// TIA Portal project "MTU_Bauteilträger(BTTR)_V16" (V16)

(* hardware
DEVICE "ET 200SP station_1"  ET 200SP-Station
   slot 0: "Rack_0"  Rack  6ES5 710-8MAx1
   slot 1: "-33K1"  CPU 1512SP F-1 PN  6ES7 512-1SK01-0AB0  V2.8
      slot 32768: "PROFINET interface_1"  X1
   slot 2: "-33K2"  DI 16x24VDC ST  6ES7 131-6BH01-0BA0  V0.0
      slot 1: "-33K2"  DI 16x24VDC ST
   slot 3: "-33K3"  DI 16x24VDC ST  6ES7 131-6BH01-0BA0  V0.0
      slot 1: "-33K3"  DI 16x24VDC ST
   slot 4: "-33K5"  DQ 4x24VDC/2A ST  6ES7 132-6BD20-0BA0  V1.1
      slot 1: "-33K5"  DQ 4x24VDC/2A ST
   slot 5: "-33K6"  DQ 4x24VDC/2A ST  6ES7 132-6BD20-0BA0  V1.1
      slot 1: "-33K6"  DQ 4x24VDC/2A ST
   slot 6: "Server module_1"  Server module  6ES7 193-6PA00-0AA0  V1.1
      slot 1: "Server module_1"  Server module
   slot 127: "BA 2xRJ45"  BA 2xRJ45  6ES7 193-6AR00-0AA0  V0.0
      slot 32769: "Port_1"  6ES7 193-6AR00-0AA0
      slot 32770: "Port_2"  6ES7 193-6AR00-0AA0
DEVICE "-55K1"  PnPn.Device
   slot 0: "Rack"  Rail  1.0
   slot 0: "pn-pn-coupler.X1"  PN/PN Coupler  6ES7 158-3AD10-0XA0  V4.2
   slot 1: "pn-pn-coupler"  PN/PN Coupler  6ES7 158-3AD10-0XA0  V4.2
   slot 127: "BA 2xRJ45"  BA 2xRJ45  6ES7 193-6AR00-0AA0  V0.0
      slot 1: "Port_1"  X1 P1 R  6ES7 193-6AR00-0AA0  V0.0
      slot 2: "Port_2"  X1 P2 R  6ES7 193-6AR00-0AA0  V0.0
   slot 127: "BA 2xRJ45"  BA 2xRJ45  6ES7 193-6AR00-0AA0  V0.0
      slot 1: "Port_1"  X2 P1 R  6ES7 193-6AR00-0AA0  V0.0
      slot 2: "Port_2"  X2 P2 R  6ES7 193-6AR00-0AA0  V0.0
*)

// ===== PLC "-33K1"  CPU 1512SP F-1 PN =====

VAR_GLOBAL   // PLC tag table "Default tag table"
   "System_Byte" AT %MB1 : Byte;
   "FirstScan" AT %M1.0 : Bool;
   "DiagStatusUpdate" AT %M1.1 : Bool;
   "AlwaysTRUE" AT %M1.2 : Bool;
   "AlwaysFALSE" AT %M1.3 : Bool;
   "System_Byte(1)" AT %MB1 : Byte;
   "Clock_Byte" AT %MB0 : Byte;
   "Clock_10Hz" AT %M0.0 : Bool;
   "Clock_5Hz" AT %M0.1 : Bool;
   "Clock_2.5Hz" AT %M0.2 : Bool;
   "Clock_2Hz" AT %M0.3 : Bool;
   "Clock_1.25Hz" AT %M0.4 : Bool;
   "Clock_1Hz" AT %M0.5 : Bool;
   "Clock_0.625Hz" AT %M0.6 : Bool;
   "Clock_0.5Hz" AT %M0.7 : Bool;
END_VAR

VAR_GLOBAL   // PLC tag table "Ausgänge"
   "O_BTTR1_UnlockComp" AT %Q1610.0 : Bool;   // Bauteilträger 1 Bauteil entriegeln (1=entriegeln)
   "O_BTTR2_UnlockComp" AT %Q1610.1 : Bool;   // Bauteilträger 2 Bauteil entriegeln (1=entriegeln)
   "O_BTTR3_UnlockComp" AT %Q1610.2 : Bool;   // Bauteilträger 3 Bauteil entriegeln (1=entriegeln)
   "O_BTTR4_UnlockComp" AT %Q1610.3 : Bool;   // Bauteilträger 4 Bauteil entriegeln (1=entriegeln)
   "O_BTTR5_UnlockComp" AT %Q1611.0 : Bool;   // Bauteilträger 5 Bauteil entriegeln (1=entriegeln)
   "O_BTTR6_UnlockComp" AT %Q1611.1 : Bool;   // Bauteilträger 6 Bauteil entriegeln (1=entriegeln)
   "A1611.2" AT %Q1611.2 : Bool;   // Reserve
   "A1611.3" AT %Q1611.3 : Bool;   // Reserve
END_VAR

VAR_GLOBAL   // PLC tag table "Eingänge"
   "I_BTTR1_CompMon" AT %I1610.0 : Bool;   // Bauteilträger 1 INS Bauteilüberwachung (0=Platz leer/1=Platz belegt)
   "I_BTTR1_CompLock_SW1" AT %I1610.1 : Bool;   // Bauteilträger 1 RM Bauteilverriegelung Schalter 1
   "I_BTTR1_CompLock_SW2" AT %I1610.2 : Bool;   // Bauteilträger 1 RM Bauteilverriegelung Schalter 2
   "E1610.3" AT %I1610.3 : Bool;   // Bauteilträger 1 Reserve
   "I_BTTR2_CompMon" AT %I1610.4 : Bool;   // Bauteilträger 2 INS Bauteilüberwachung (0=Platz leer/1=Platz belegt)
   "I_BTTR2_CompLock_SW1" AT %I1610.5 : Bool;   // Bauteilträger 2 RM Bauteilverriegelung Schalter 1
   "I_BTTR2_CompLock_SW2" AT %I1610.6 : Bool;   // Bauteilträger 2 RM Bauteilverriegelung Schalter 2
   "E1610.7" AT %I1610.7 : Bool;   // Bauteilträger 2 Reserve
   "I_BTTR3_CompMon" AT %I1611.0 : Bool;   // Bauteilträger 3 INS Bauteilüberwachung (0=Platz leer/1=Platz belegt)
   "I_BTTR3_CompLock_SW1" AT %I1611.1 : Bool;   // Bauteilträger 3 RM Bauteilverriegelung Schalter 1
   "I_BTTR3_CompLock_SW2" AT %I1611.2 : Bool;   // Bauteilträger 3 RM Bauteilverriegelung Schalter 2
   "E1611.3" AT %I1611.3 : Bool;   // Bauteilträger 3 Reserve
   "I_BTTR4_CompMon" AT %I1611.4 : Bool;   // Bauteilträger 4 INS Bauteilüberwachung (0=Platz leer/1=Platz belegt)
   "I_BTTR4_CompLock_SW1" AT %I1611.5 : Bool;   // Bauteilträger 4 RM Bauteilverriegelung Schalter 1
   "I_BTTR4_CompLock_SW2" AT %I1611.6 : Bool;   // Bauteilträger 4 RM Bauteilverriegelung Schalter 2
   "E1611.7" AT %I1611.7 : Bool;   // Bauteilträger 4 Reserve
   "I_BTTR5_CompMon" AT %I1612.0 : Bool;   // Bauteilträger 5 INS Bauteilüberwachung (0=Platz leer/1=Platz belegt)
   "I_BTTR5_CompLock_SW1" AT %I1612.1 : Bool;   // Bauteilträger 5 RM Bauteilverriegelung Schalter 1
   "I_BTTR5_CompLock_SW2" AT %I1612.2 : Bool;   // Bauteilträger 5 RM Bauteilverriegelung Schalter 2
   "E1612.3" AT %I1612.3 : Bool;   // Bauteilträger 5 Reserve
   "I_BTTR6_CompMon" AT %I1612.4 : Bool;   // Bauteilträger 6 INS Bauteilüberwachung (0=Platz leer/1=Platz belegt)
   "I_BTTR6_CompLock_SW1" AT %I1612.5 : Bool;   // Bauteilträger 6 RM Bauteilverriegelung Schalter 1
   "I_BTTR6_CompLock_SW2" AT %I1612.6 : Bool;   // Bauteilträger 6 RM Bauteilverriegelung Schalter 2
   "E1612.7" AT %I1612.7 : Bool;   // Bauteilträger 6 Reserve
   "I_TankLevel_75" AT %I1613.0 : Bool;   // Tanküberwachung Füllstand >=75% (0=>=75%/1=<=75%)
   "E1613.1" AT %I1613.1 : Bool;   // Tanküberwachung Füllstand >=75% Reserve
   "I_TankLevel_100" AT %I1613.2 : Bool;   // Tanküberwachung Füllstand >=100% (0=>=100%/1=<=100%)
   "E1613.3" AT %I1613.3 : Bool;   // Tanküberwachung Füllstand >=100% Reserve
   "E1613.4" AT %I1613.4 : Bool;   // Reserve
   "E1613.5" AT %I1613.5 : Bool;   // Reserve
   "E1613.6" AT %I1613.6 : Bool;   // Reserve
   "E1613.7" AT %I1613.7 : Bool;   // Reserve
END_VAR

TYPE "UDT_BTTR"
   STRUCT
      ID : DInt;   // Aktuelle Nummer vom Bild
      ESF_ID : DInt;   // Nummer für die Textliste für Zylindernamen
      ESF_Nr : DInt;   // angewählte ESF in der HMI
      Ctrl : Struct
         Unlock : Bool;   // Command to unlock
         Reset_error : Bool;   // Command to reset error
      END_STRUCT;
      Status : Struct
         UnLocked : Bool;   // State (1- unlocked, 0 - locked)
         ErrorBit : Bool;   // Error flag
         ErrorByte : Byte;   // Error type
      END_STRUCT;
   END_STRUCT;
END_TYPE

TYPE "UDT_FM_Bits"
VERSION : 0.1
   STRUCT
      SM : Array[1..2048] of Bool;
   END_STRUCT;
END_TYPE

// folder: Sensor

TYPE "UDT_T_Sensor"
   STRUCT
      Rohsignal : Bool;   // Direkt vom Eingangsignal
      Frei : Bool;   // Sensor frei
      Belegt : Bool;   // Sensor belegt
      T_Frei : Bool;   // Sensor mit T-Zeit frei
      T_Belegt : Bool;   // Senssor mit T-zeit belegt
      T_Dauer_Belegt : Bool;
      Fehler : Bool;   // Fehler aktiv
      Status : Byte;   // 0 = OK 1 = nicht frei 2=nicht belegt
      Temp_Fehler : Struct   // Fehler generieren und wird automatisch im Sensorbaustein zurückgesetzt
         Nicht_frei : Bool;   // Fehler Sensor nicht frei
         Nicht_belegt : Bool;   // Fehler Sensor nicht belegt
      END_STRUCT;
      Setup : Struct
         T_Frei : Time := T#100MS;
         T_Belegt : Time := T#100MS;
         T_Dauer : Time := T#10S;
         Typ : Bool;   // 0 = S 1 = Ö
         Mode : Byte;
      END_STRUCT;
   END_STRUCT;
END_TYPE

TYPE "UDTFltFbStructSeqSK"
   STRUCT
      Aktiv : Byte;   // 1=Aktiv
      Msg : Byte;   // 1=FLT 2=Warn 10=Clear
      StepNo : Int;
      FltID : DInt;
      DeviceID : DInt;
      Station : DInt;
      DeviceText : String[20];
   END_STRUCT;
END_TYPE

// folder: DBs

DATA_BLOCK "DB_Sensors"   // DB1
{ S7_Optimized_Access := 'TRUE' }
VERSION : 0.1
   VAR
      "Sens_BTTR1-11BG1" : "UDT_T_Sensor";   // Bauteilträger 1 INS Bauteilüberwachung (0=Platz leer/1=Platz belegt)
      "Sens_BTTR2-13BG1" : "UDT_T_Sensor";   // Bauteilträger 2 INS Bauteilüberwachung (0=Platz leer/1=Platz belegt)
      "Sens_BTTR3-15BG1" : "UDT_T_Sensor";   // Bauteilträger 3 INS Bauteilüberwachung (0=Platz leer/1=Platz belegt)
      "Sens_BTTR4-17BG1" : "UDT_T_Sensor";   // Bauteilträger 4 INS Bauteilüberwachung (0=Platz leer/1=Platz belegt)
      "Sens_BTTR5-19BG1" : "UDT_T_Sensor";   // Bauteilträger 5 INS Bauteilüberwachung (0=Platz leer/1=Platz belegt)
      "Sens_BTTR6-21BG1" : "UDT_T_Sensor";   // Bauteilträger 6 INS Bauteilüberwachung (0=Platz leer/1=Platz belegt)
      "Sens_UGBTTR-23A1" : "UDT_T_Sensor";   // Tank Untergestell Füllstand >=75%
      "Sens_UGBTTR-23A2" : "UDT_T_Sensor";   // Tank Untergestell Füllstand >=100%
   END_VAR
BEGIN
END_DATA_BLOCK

DATA_BLOCK "DB_M1_SM"   // DB2
{ S7_Optimized_Access := 'TRUE' }
VERSION : 0.1
   VAR
      SM : "UDT_FM_Bits";
      SM_Byte : Array[1..2048] of Byte;
      SM_DInt : Array[1..2048] of DInt;
      SM_Word_Komm : Array[1..100] of Word;
   END_VAR
BEGIN
END_DATA_BLOCK

DATA_BLOCK "DB_BTTR"   // DB4
{ S7_Optimized_Access := 'TRUE' }
VERSION : 0.1
   VAR
      "BTTR1-11K1" : "UDT_BTTR";   // elektr. mag. Verriegelungseinheit Bauteilträger1
      "BTTR2-13K1" : "UDT_BTTR";   // elektr. mag. Verriegelungseinheit Bauteilträger2
      "BTTR3-15K1" : "UDT_BTTR";   // elektr. mag. Verriegelungseinheit Bauteilträger3
      "BTTR4-17K1" : "UDT_BTTR";   // elektr. mag. Verriegelungseinheit Bauteilträger4
      "BTTR5-19K1" : "UDT_BTTR";   // elektr. mag. Verriegelungseinheit Bauteilträger5
      "BTTR6-21K1" : "UDT_BTTR";   // elektr. mag. Verriegelungseinheit Bauteilträger6
   END_VAR
BEGIN
END_DATA_BLOCK

DATA_BLOCK "DB_SPS-BTTR_ProfinetComm"   // DB6
{ S7_Optimized_Access := 'TRUE' }
VERSION : 0.1
   VAR
      DataIn : Struct   // XXX_to_SPS(BTTR/MAG)
         robotSafeArea : Bool;   // Robot out of magazin-area
         enableMagazinMotion : Bool;   // Magazin allowed to turn
         requestIdentification : Bool;   // Identification of loaded parts requested
         robotDoor1Open : Bool;   // Command to open robot-door amr
         robotDoor1Close : Bool;   // Command to close robot-door amr
         robotDoor2Open : Bool;   // Command to open robot-door fix
         robotDoor2Close : Bool;   // Command to close robot-door fix
         "Bit0.7" : Bool;
         requestUndock : Bool;   // Request from AMR to undock
         requestCommunication : Bool;   // Request from PN-Station to take masterpart on communication
         "Bit1.2" : Bool;
         "Bit1.3" : Bool;
         "Bit1.4" : Bool;
         "Bit1.5" : Bool;
         unlockBTTRRequest : Bool;   // Request from Robot to unlock BTTR
         resetBTTRerror : Bool;   // To reset BTTR errors
         requestPlace : UInt;   // Byte2 - Requested place to move
         requestLevel : UInt;   // Byte4 - Requested level for postion to move
         requestPosition : UInt;   // Byte6 - Requested positin to move
         requestSide : UInt;   // Byte8 - Requested place to move on requested side
         Byte10 : Byte;   // Byte10
         Byte11_1 : Byte;   // Byte11
         Byte12_1 : Byte;   // Byte12
         Byte13_1 : Byte;   // Byte13
         Byte14_1 : Byte;   // Byte14
         Byte15_1 : Byte;   // Byte15
         Byte16_1 : Byte;   // Byte16
         Byte17_1 : Byte;   // Byte17
         Byte18_1 : Byte;   // Byte18
         Byte19_1 : Byte;   // Byte19
         Byte20_1 : Byte;   // Byte20
         Byte21_1 : Byte;   // Byte21
         Byte22_1 : Byte;   // Byte22
         Byte23_1 : Byte;   // Byte23
         Byte24_1 : Byte;   // Byte24
         Byte25_1 : Byte;   // Byte25
         Byte26_1 : Byte;   // Byte26
         Byte27_1 : Byte;   // Byte27
         Byte28_1 : Byte;   // Byte28
         Byte29_1 : Byte;   // Byte29
         Byte30_1 : Byte;   // Byte30
         Byte31_1 : Byte;   // Byte10
         Byte32_1 : Byte;   // Byte10
         Byte33_1 : Byte;   // Byte10
         Byte34_1 : Byte;   // Byte10
         Byte35_1 : Byte;   // Byte10
         Byte36_1 : Byte;   // Byte10
         Byte37_1 : Byte;   // Byte10
         Byte38_1 : Byte;   // Byte10
         Byte39_1 : Byte;   // Byte10
         Byte40_1 : Byte;   // Byte10
         Byte41_1 : Byte;   // Byte10
         Byte42_1 : Byte;   // Byte10
         Byte43_1 : Byte;   // Byte10
         Byte44_1 : Byte;   // Byte10
         Byte45_1 : Byte;   // Byte10
         Byte46_1 : Byte;   // Byte10
         Byte47_1 : Byte;   // Byte10
         Byte48_1 : Byte;   // Byte10
         Byte49_1 : Byte;   // Byte10
         Byte50_1 : Byte;   // Byte10
         Byte51_1 : Byte;   // Byte10
         Byte52_1 : Byte;   // Byte10
         Byte53_1 : Byte;   // Byte10
         Byte54_1 : Byte;   // Byte10
         Byte55_1 : Byte;   // Byte10
         Byte56_1 : Byte;   // Byte10
         Byte57_1 : Byte;   // Byte10
         Byte58_1 : Byte;   // Byte10
         Byte59_1 : Byte;   // Byte10
         Byte60_1 : Byte;   // Byte10
         Byte61_1 : Byte;   // Byte10
         Byte62_1 : Byte;   // Byte10
         Byte63_1 : Byte;   // Byte10
      END_STRUCT;
      DataOut : Struct   // SPS(BTTR/MAG)_to_XXX
         placeDone : Bool;   // Signal indicating moving on requested place done
         enableRobotAccess1 : Bool;   // Signal indicating access for robot amr enabled
         enableRobotAccess2 : Bool;   // Signal indicating access for robot fix enabled
         "Bit0.3" : Bool;
         "Bit0.4" : Bool;
         "Bit0.5" : Bool;
         "Bit0.6" : Bool;
         "Bit0.7" : Bool;
         readyForUndock : Bool;   // Signal indicating magazin is ready to undock
         "Bit1.1" : Bool;
         "Bit1.2" : Bool;
         "Bit1.3" : Bool;
         "Bit1.4" : Bool;
         "Bit1.5" : Bool;
         "Bit1.6" : Bool;
         "Bit1.7" : Bool;
         state : Word;   // Byte2-3
         errorIndication : Word;   // Byte4-5
         placeNbrAct : UInt;   // Byte6-7
         zlr : String[16];   // Byte8-25 - serial number of PLC
         sanr : String[16] := 'BTTR';   // Byte26-43
         InductiveBTTRsensor : Word;   // Byte44-45 (six first bits for six sensors)
         BTTRerror : Word;   // Byte46-47 (six first bits for six BTTR)
         BTTRunlocked : Bool;   // Bit48.0 (BTTR1…6 are unlocked )
         level_75 : Bool;   // Bit48.1 (Tank monitoring level> = 75%)
         level_100 : Bool;   // Bit48.2 (Tank monitoring level> = 100%)
         "Bit48.3" : Bool;
         "Bit48.4" : Bool;
         "Bit48.5" : Bool;
         "Bit48.6" : Bool;
         "Bit48.7" : Bool;
         Byte49 : Byte;
         Byte50 : Byte;
         Byte51 : Byte;
         Byte52 : Byte;
         Byte53 : Byte;
         Byte54 : Byte;
         Byte55 : Byte;
         Byte56 : Byte;
         Byte57 : Byte;
         Byte58 : Byte;
         Byte59 : Byte;
         Byte60 : Byte;
         Byte61 : Byte;
         Byte62 : Byte;
         Byte63 : Byte;
      END_STRUCT;
      StatusRead : DWord;
      StatusWrite : DWord;
      LengthRead : Int;
   END_VAR
BEGIN
END_DATA_BLOCK

// folder: Instances

DATA_BLOCK "Sensors_DB"   // DB3
{ S7_Optimized_Access := 'TRUE' }
VERSION : 0.1
// stored: InstanceOfName ESF_Sensors
"ESF_Sensors"
BEGIN
END_DATA_BLOCK

DATA_BLOCK "ESF_BTTR_DB"   // DB5
{ S7_Optimized_Access := 'TRUE' }
VERSION : 0.1
// stored: InstanceOfName ESF_BTTR
"ESF_BTTR"
BEGIN
END_DATA_BLOCK

DATA_BLOCK "BTTR_Control_DB"   // DB7
{ S7_Optimized_Access := 'TRUE' }
VERSION : 0.1
// stored: InstanceOfName BTTR_Control
"BTTR_Control"
BEGIN
END_DATA_BLOCK

// folder: (top level)

FUNCTION_BLOCK "ESF_Sensors"   // FB1, SCL
{ S7_Optimized_Access := 'TRUE' }
VERSION : 0.1
   VAR
      "Sens_BTTR1-11BG1" : "FB_T_Sensor";
      "Sens_BTTR2-13BG1" : "FB_T_Sensor";
      "Sens_BTTR3-15BG1" : "FB_T_Sensor";
      "Sens_BTTR4-17BG1" : "FB_T_Sensor";
      "Sens_BTTR5-19BG1" : "FB_T_Sensor";
      "Sens_BTTR6-21BG1" : "FB_T_Sensor";
      "Sens_UGBTTR-23A1" : "FB_T_Sensor";
      "Sens_UGBTTR-23A2" : "FB_T_Sensor";
   END_VAR
BEGIN
   (*##############################################################################################################################*)
   (*                                                 FunctionBlock Description                                                    *)
   (*##############################################################################################################################*)
   (*################################################################################################################################
   Created by: preccon Robotics
   Department: 
   Creator: d.shulgin
   Creation Date: 2021-09-24
   Version: V1.0.0.0
   Function Description:
       Inputs:
           --NONE--
           Description in IO table
       Outputs:
           --NONE--
           Description in IO table
       Function:
           Creating sensors instances  

   Last Changed:
       2021-09-24 d.shulgin: V1.0.0.0 Created FunctionBlock

   ################################################################################################################################*)



   REGION Bauteilträger 1 INS Bauteilüberwachung
      #"Sens_BTTR1-11BG1"(E_Sensor:="I_BTTR1_CompMon",
                          SensorMode:=0,
                          Error => "DB_M1_SM".SM.SM[501],//flag of error [size - bool]
                          "ErrorState" => "DB_M1_SM".SM_Byte[501],//type of error [size - byte]
                          Sensor:="DB_Sensors"."Sens_BTTR1-11BG1");
   END_REGION

   REGION Bauteilträger 2 INS Bauteilüberwachung
       #"Sens_BTTR2-13BG1"(E_Sensor:="I_BTTR2_CompMon",
                           SensorMode:=0,
                           Error => "DB_M1_SM".SM.SM[502],
                           "ErrorState" => "DB_M1_SM".SM_Byte[502],
                           Sensor:="DB_Sensors"."Sens_BTTR2-13BG1");
   END_REGION

   REGION Bauteilträger 3 INS Bauteilüberwachung
       #"Sens_BTTR3-15BG1"(E_Sensor:="I_BTTR3_CompMon",
                           SensorMode:=0,
                           Error => "DB_M1_SM".SM.SM[503],
                           "ErrorState" => "DB_M1_SM".SM_Byte[503],
                           Sensor:="DB_Sensors"."Sens_BTTR3-15BG1");
   END_REGION

   REGION Bauteilträger 4 INS Bauteilüberwachung
       #"Sens_BTTR4-17BG1"(E_Sensor:="I_BTTR4_CompMon",
                           SensorMode:=0,
                           Error => "DB_M1_SM".SM.SM[504],
                           "ErrorState" => "DB_M1_SM".SM_Byte[504],
                           Sensor:="DB_Sensors"."Sens_BTTR4-17BG1");
   END_REGION

   REGION Bauteilträger 5 INS Bauteilüberwachung
       #"Sens_BTTR5-19BG1"(E_Sensor:="I_BTTR5_CompMon",
                           SensorMode:=0,
                           Error => "DB_M1_SM".SM.SM[505],
                           "ErrorState" => "DB_M1_SM".SM_Byte[505],
                           Sensor:="DB_Sensors"."Sens_BTTR5-19BG1");
   END_REGION

   REGION Bauteilträger 6 INS Bauteilüberwachung
       #"Sens_BTTR6-21BG1"(E_Sensor:="I_BTTR6_CompMon",
                           SensorMode:=0,
                           Error => "DB_M1_SM".SM.SM[506],
                           "ErrorState" => "DB_M1_SM".SM_Byte[506],
                           Sensor:="DB_Sensors"."Sens_BTTR6-21BG1");
   END_REGION


   REGION Tanküberwachung Füllstand >=75% (0=>=75%/1=<=75%)
       #"Sens_UGBTTR-23A1"(E_Sensor := "I_TankLevel_75",
                           SensorMode := 0,
                           Error => "DB_M1_SM".SM.SM[507],
                           "ErrorState" => "DB_M1_SM".SM_Byte[507],
                           Sensor := "DB_Sensors"."Sens_UGBTTR-23A1");
   END_REGION

   REGION Tanküberwachung Füllstand >=100% (0=>=100%/1=<=100%)
       #"Sens_UGBTTR-23A2"(E_Sensor:="I_TankLevel_100",
                           SensorMode:=0,
                           Error => "DB_M1_SM".SM.SM[508],
                           "ErrorState" => "DB_M1_SM".SM_Byte[508],
                           Sensor:="DB_Sensors"."Sens_UGBTTR-23A2");
   END_REGION
END_FUNCTION_BLOCK

FUNCTION_BLOCK "ESF_BTTR"   // FB3, SCL
{ S7_Optimized_Access := 'TRUE' }
VERSION : 0.1
   VAR
      BTTR1 : "FB_BTTR_Ctrl";
      BTTR2 : "FB_BTTR_Ctrl";
      BTTR3 : "FB_BTTR_Ctrl";
      BTTR4 : "FB_BTTR_Ctrl";
      BTTR5 : "FB_BTTR_Ctrl";
      BTTR6 : "FB_BTTR_Ctrl";
   END_VAR
BEGIN
   (*##############################################################################################################################*)
   (*                                                 FunctionBlock Description                                                    *)
   (*##############################################################################################################################*)
   (*################################################################################################################################
   Created by: preccon Robotics
   Department: 
   Creator: d.shulgin
   Creation Date: 2021-09-24
   Version: V1.0.0.0
   Function Description:
       Inputs:
           --NONE--
           Description in IO table
       Outputs:
           --NONE--
           Description in IO table
       Function:
           Creating 6 instances for 6 BTTR units 

   Last Changed:
       2021-09-24 d.shulgin: V1.0.0.0 Created FunctionBlock

   ################################################################################################################################*)


   REGION BTTR1-11K1
   #BTTR1(Verr_Unlock:=FALSE,
          Freigabe:=TRUE,
          E_Schalter1:="I_BTTR1_CompLock_SW1",
          E_Schalter2:="I_BTTR1_CompLock_SW2",
          A_BTTR_Unlock=>"O_BTTR1_UnlockComp",
          BTTR:="DB_BTTR"."BTTR1-11K1");

   END_REGION

   REGION BTTR2-13K1
       #BTTR2(Verr_Unlock:=FALSE,
              Freigabe:=TRUE,
              E_Schalter1:="I_BTTR2_CompLock_SW1",
              E_Schalter2:="I_BTTR2_CompLock_SW2",
              A_BTTR_Unlock=>"O_BTTR2_UnlockComp",
              BTTR:="DB_BTTR"."BTTR2-13K1");

   END_REGION

   REGION BTTR3-15K1
       #BTTR3(Verr_Unlock:=FALSE,
              Freigabe:=TRUE,
              E_Schalter1:="I_BTTR3_CompLock_SW1",
              E_Schalter2:="I_BTTR3_CompLock_SW2",
              A_BTTR_Unlock=>"O_BTTR3_UnlockComp",
              BTTR:="DB_BTTR"."BTTR3-15K1");

   END_REGION

   REGION BTTR4-17K1
       #BTTR4(Verr_Unlock:=FALSE,
              Freigabe:=TRUE,
              E_Schalter1:="I_BTTR4_CompLock_SW1",
              E_Schalter2:="I_BTTR4_CompLock_SW2",
              A_BTTR_Unlock=>"O_BTTR4_UnlockComp",
              BTTR:="DB_BTTR"."BTTR4-17K1");

   END_REGION

   REGION BTTR5-19K1
       #BTTR5(Verr_Unlock:=FALSE,
              Freigabe:=TRUE,
              E_Schalter1:="I_BTTR5_CompLock_SW1",
              E_Schalter2:="I_BTTR5_CompLock_SW2",
              A_BTTR_Unlock=>"O_BTTR5_UnlockComp",
              BTTR:="DB_BTTR"."BTTR5-19K1");

   END_REGION

   REGION BTTR6-21K1
       #BTTR6(Verr_Unlock:=FALSE,
              Freigabe:=TRUE,
              E_Schalter1:="I_BTTR6_CompLock_SW1",
              E_Schalter2:="I_BTTR6_CompLock_SW2",
              A_BTTR_Unlock=>"O_BTTR6_UnlockComp",
              BTTR:="DB_BTTR"."BTTR6-21K1");

   END_REGION
END_FUNCTION_BLOCK

FUNCTION_BLOCK "BTTR_Control"   // FB4, SCL
{ S7_Optimized_Access := 'TRUE' }
VERSION : 0.1
   VAR
      GETIO_Instance : GETIO;   // Profinet IO interface READ
      SETIO_Instance : SETIO;   // Profinet IO interface WRITE
      GET_IM_DATA_Instance : Get_IM_Data;
      bGetImDataDONE : Bool;
      imData : IM0_Data;
   END_VAR
BEGIN
   (*##############################################################################################################################*)
   (*                                                 FunctionBlock Description                                                    *)
   (*##############################################################################################################################*)
   (*################################################################################################################################
   Created by: preccon Robotics
   Department: 
   Creator: d.shulgin
   Creation Date: 2021-09-24
   Version: V1.0.0.0
   Function Description:
       Inputs:
           --NONE--
           Description in IO table
       Outputs:
           --NONE--
           Description in IO table
       Function:
           Read/Write profinet IO-signals beatween BTTR and AMR CS9 

   Last Changed:
       2021-09-24 d.shulgin: V1.0.0.0 Created FunctionBlock
       2021-10-04 d.shulgin: inverse signals from sensors "Bauteilträger Bauteilüberwachung"
       2021-10-06 d.shulgin: Updating signals in "DB_SPS-BTTR_ProfinetComm[DB6]"
       2021-10-08 d.shulgin: Adding reading serial number function
       2021-10-12 d.shulgin: Adding pn-pn Coupler
       2021-10-12 d.shulgin: Updating signals in "DB_SPS-BTTR_ProfinetComm[DB6]"

   ################################################################################################################################*)



   REGION Init
       //Read PLC serial number
       #GET_IM_DATA_Instance(LADDR:="Local",
                             IM_TYPE:=0,
                             DONE=>#bGetImDataDONE,
                             DATA:=#imData);

       IF #bGetImDataDONE THEN
           "DB_SPS-BTTR_ProfinetComm".DataOut.zlr:=#imData.Serial_Number;
       END_IF;
   END_REGION


   REGION READ Profinet IO signals
       #GETIO_Instance(ID:="pn-pn-coupler_X1~PROFINET_interface_X1~Rob_toPLC",
                       STATUS=>"DB_SPS-BTTR_ProfinetComm".StatusRead,
                       LEN=>"DB_SPS-BTTR_ProfinetComm".LengthRead,
                       INPUTS:="DB_SPS-BTTR_ProfinetComm".DataIn);

   END_REGION


   REGION Control BTTR
       "DB_BTTR"."BTTR1-11K1".Ctrl.Unlock := "DB_SPS-BTTR_ProfinetComm".DataIn.unlockBTTRRequest;
       "DB_BTTR"."BTTR2-13K1".Ctrl.Unlock := "DB_SPS-BTTR_ProfinetComm".DataIn.unlockBTTRRequest;
       "DB_BTTR"."BTTR3-15K1".Ctrl.Unlock := "DB_SPS-BTTR_ProfinetComm".DataIn.unlockBTTRRequest;
       "DB_BTTR"."BTTR4-17K1".Ctrl.Unlock := "DB_SPS-BTTR_ProfinetComm".DataIn.unlockBTTRRequest;
       "DB_BTTR"."BTTR5-19K1".Ctrl.Unlock := "DB_SPS-BTTR_ProfinetComm".DataIn.unlockBTTRRequest;
       "DB_BTTR"."BTTR6-21K1".Ctrl.Unlock := "DB_SPS-BTTR_ProfinetComm".DataIn.unlockBTTRRequest;

       //BTTR State - Lock/unLock
       IF "DB_BTTR"."BTTR1-11K1".Status.UnLocked AND
           "DB_BTTR"."BTTR2-13K1".Status.UnLocked AND
           "DB_BTTR"."BTTR3-15K1".Status.UnLocked AND
           "DB_BTTR"."BTTR4-17K1".Status.UnLocked AND
           "DB_BTTR"."BTTR5-19K1".Status.UnLocked AND
           "DB_BTTR"."BTTR6-21K1".Status.UnLocked THEN
           "DB_SPS-BTTR_ProfinetComm".DataOut.BTTRunlocked := TRUE;
       ELSE
           "DB_SPS-BTTR_ProfinetComm".DataOut.BTTRunlocked := FALSE;
       END_IF;


   END_REGION

   REGION Sensors conditions
       "DB_SPS-BTTR_ProfinetComm".DataOut.InductiveBTTRsensor.%X0 := NOT "DB_Sensors"."Sens_BTTR1-11BG1".Belegt;
       "DB_SPS-BTTR_ProfinetComm".DataOut.InductiveBTTRsensor.%X1 := NOT "DB_Sensors"."Sens_BTTR2-13BG1".Belegt;
       "DB_SPS-BTTR_ProfinetComm".DataOut.InductiveBTTRsensor.%X2 := NOT "DB_Sensors"."Sens_BTTR3-15BG1".Belegt;
       "DB_SPS-BTTR_ProfinetComm".DataOut.InductiveBTTRsensor.%X3 := NOT "DB_Sensors"."Sens_BTTR4-17BG1".Belegt;
       "DB_SPS-BTTR_ProfinetComm".DataOut.InductiveBTTRsensor.%X4 := NOT "DB_Sensors"."Sens_BTTR5-19BG1".Belegt;
       "DB_SPS-BTTR_ProfinetComm".DataOut.InductiveBTTRsensor.%X5 := NOT "DB_Sensors"."Sens_BTTR6-21BG1".Belegt;

       "DB_SPS-BTTR_ProfinetComm".DataOut.level_75 := "DB_Sensors"."Sens_UGBTTR-23A1".Belegt;
       "DB_SPS-BTTR_ProfinetComm".DataOut.level_100 := "DB_Sensors"."Sens_UGBTTR-23A2".Belegt;

   END_REGION

   REGION BTTR-error
       REGION reset BTTR-error
           IF "DB_SPS-BTTR_ProfinetComm".DataIn.resetBTTRerror THEN
               "DB_BTTR"."BTTR1-11K1".Status.ErrorBit := FALSE;
               "DB_BTTR"."BTTR2-13K1".Status.ErrorBit := FALSE;
               "DB_BTTR"."BTTR3-15K1".Status.ErrorBit := FALSE;
               "DB_BTTR"."BTTR4-17K1".Status.ErrorBit := FALSE;
               "DB_BTTR"."BTTR5-19K1".Status.ErrorBit := FALSE;
               "DB_BTTR"."BTTR6-21K1".Status.ErrorBit := FALSE;

               "DB_BTTR"."BTTR1-11K1".Status.ErrorByte := 0;
               "DB_BTTR"."BTTR2-13K1".Status.ErrorByte := 0;
               "DB_BTTR"."BTTR3-15K1".Status.ErrorByte := 0;
               "DB_BTTR"."BTTR4-17K1".Status.ErrorByte := 0;
               "DB_BTTR"."BTTR5-19K1".Status.ErrorByte := 0;
               "DB_BTTR"."BTTR6-21K1".Status.ErrorByte := 0;
           END_IF;
       END_REGION


       "DB_SPS-BTTR_ProfinetComm".DataOut.BTTRerror.%X0:="DB_BTTR"."BTTR1-11K1".Status.ErrorBit;
       "DB_SPS-BTTR_ProfinetComm".DataOut.BTTRerror.%X1 := "DB_BTTR"."BTTR2-13K1".Status.ErrorBit;
       "DB_SPS-BTTR_ProfinetComm".DataOut.BTTRerror.%X2 := "DB_BTTR"."BTTR3-15K1".Status.ErrorBit;
       "DB_SPS-BTTR_ProfinetComm".DataOut.BTTRerror.%X3 := "DB_BTTR"."BTTR4-17K1".Status.ErrorBit;
       "DB_SPS-BTTR_ProfinetComm".DataOut.BTTRerror.%X4 := "DB_BTTR"."BTTR5-19K1".Status.ErrorBit;
       "DB_SPS-BTTR_ProfinetComm".DataOut.BTTRerror.%X5 := "DB_BTTR"."BTTR6-21K1".Status.ErrorBit;
   END_REGION

   REGION WRITE Profinet IO signals
       #SETIO_Instance(ID:="pn-pn-coupler_X1~PROFINET_interface_X1~PLC_toROB",
                       STATUS=>"DB_SPS-BTTR_ProfinetComm".StatusWrite,
                       OUTPUTS:="DB_SPS-BTTR_ProfinetComm".DataOut);

   END_REGION
END_FUNCTION_BLOCK

ORGANIZATION_BLOCK "Main"   // OB1, LAD, ProgramCycle
TITLE = "Main Program Sweep (Cycle)"
{ S7_Optimized_Access := 'TRUE' }
VERSION : 0.1
   VAR_INPUT
      Initial_Call : Bool;   // Initial call of this OB
      Remanence : Bool;   // =True, if remanent data are available
   END_VAR
BEGIN

REGION Network 1: Sensors reading
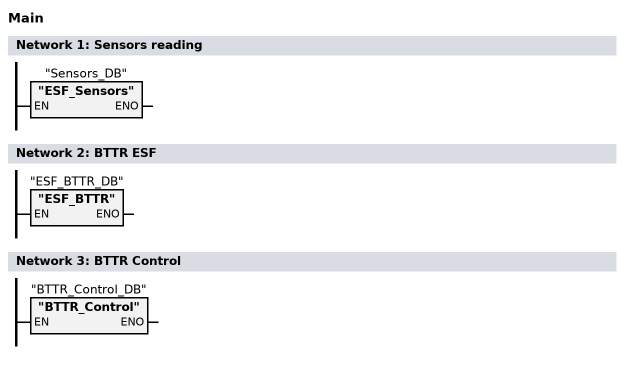
   RUNG wire#powerrail
      "Sensors_DB"()
   END_RUNG
   // the same network as SCL:
   "Sensors_DB"();   // "ESF_Sensors"
END_REGION

REGION Network 2: BTTR ESF
   RUNG wire#powerrail
      "ESF_BTTR_DB"()
   END_RUNG
   // the same network as SCL:
   "ESF_BTTR_DB"();   // "ESF_BTTR"
END_REGION

REGION Network 3: BTTR Control
   RUNG wire#powerrail
      "BTTR_Control_DB"()
   END_RUNG
   // the same network as SCL:
   "BTTR_Control_DB"();   // "BTTR_Control"
END_REGION
END_ORGANIZATION_BLOCK

// folder: SUB

FUNCTION_BLOCK "FB_BTTR_Ctrl"   // FB2, SCL
{ S7_Optimized_Access := 'TRUE' }
VERSION : 0.1
   VAR_INPUT
      Verr_Unlock : Bool;   // Interlock for Unlock
      Freigabe : Bool;
      E_Schalter1 : Bool;   // Feedback Signal from Schalter1
      E_Schalter2 : Bool;   // Feedback Signal from Schalter2
      ErrorTime : Time := T#2S;   // Time out for error
   END_VAR
   VAR_OUTPUT
      A_BTTR_Unlock : Bool;   // Signal to Unlock BTTR (true - unlock)
   END_VAR
   VAR_IN_OUT
      BTTR : "UDT_BTTR";   // Instance of unit
   END_VAR
   VAR
      T_Error : TON_TIME;   // Timer for error monitoring
   END_VAR
   VAR_TEMP
      TempBTTR : "UDT_BTTR";   // Temp instance of unit
      TempError : Bool;   // Temp error flag
   END_VAR
BEGIN
   (*##############################################################################################################################*)
   (*                                                 FunctionBlock Description                                                    *)
   (*##############################################################################################################################*)
   (*################################################################################################################################
   Created by: preccon Robotics
   Department: 
   Creator: d.shulgin
   Creation Date: 2021-09-24
   Version: V1.0.0.0
   Function Description:
       Inputs:
           --NONE--
           Description in IO table
       Outputs:
           --NONE--
           Description in IO table
       Function:
           Control unit BTTR (lock/unlock, error messages, state)

   Last Changed:
       2021-09-24 d.shulgin: V1.0.0.0 Created FunctionBlock

   ################################################################################################################################*)


   REGION Init

   END_REGION

   REGION Read Data
       #TempBTTR := #BTTR;
   END_REGION

   REGION BTTR STATUS (error+state)
       IF #TempBTTR.Ctrl.Unlock = FALSE AND (NOT #E_Schalter1 =TRUE) AND (NOT #E_Schalter2 = TRUE) THEN
           #TempError := TRUE;
           #TempBTTR.Status.ErrorByte := 1;
       END_IF;

       IF #TempBTTR.Ctrl.Unlock = TRUE AND (NOT #E_Schalter1=FALSE ) AND (NOT #E_Schalter2 = FALSE) THEN
           #TempError := TRUE;
           #TempBTTR.Status.ErrorByte := 2;
       END_IF;

       IF (#TempBTTR.Ctrl.Unlock = FALSE AND #E_Schalter1 = TRUE AND #E_Schalter2 = TRUE) OR
           (#TempBTTR.Ctrl.Unlock = TRUE AND #E_Schalter1 = FALSE AND #E_Schalter2 = FALSE) THEN
           #TempError := FALSE;
           #TempBTTR.Status.ErrorByte := 0;
       END_IF;

       #T_Error(IN := #TempError, //start timer
                PT := #ErrorTime);

       IF  #TempError = FALSE THEN
           #TempBTTR.Status.ErrorBit := FALSE;
           #TempBTTR.Status.ErrorByte := 0;

           //State BTTR (Locked/Unlocked)
           IF #TempBTTR.Ctrl.Unlock = TRUE AND (#E_Schalter1 = #E_Schalter2 = FALSE) THEN
               #TempBTTR.Status.UnLocked := TRUE;
           ELSIF #TempBTTR.Ctrl.Unlock = FALSE AND (#E_Schalter1 = #E_Schalter2 = TRUE) THEN
               #TempBTTR.Status.UnLocked := FALSE;
           END_IF;

       ELSIF #T_Error.Q AND #TempError = TRUE THEN
           #TempBTTR.Status.ErrorBit := TRUE;
       END_IF;

   END_REGION

   REGION Ctrl BTTR
       IF NOT #Verr_Unlock THEN
           IF (NOT #TempBTTR.Status.ErrorBit) AND #TempBTTR.Ctrl.Unlock THEN
               #A_BTTR_Unlock := TRUE;
           END_IF;
           IF NOT #TempBTTR.Ctrl.Unlock THEN
               #A_BTTR_Unlock := FALSE;
           END_IF;
       ELSE
           #A_BTTR_Unlock := FALSE;
       END_IF;
   END_REGION

   REGION Write Data
       #BTTR.Status := #TempBTTR.Status;

   END_REGION
END_FUNCTION_BLOCK

FUNCTION_BLOCK "FB_T_Sensor"   // FB134, SCL
{ S7_Optimized_Access := 'TRUE' }
VERSION : 0.1
   VAR_INPUT
      E_Sensor : Bool;   // Eingang vom Sensor
      SensorMode : Bool;   // Sensor frei; 0= Schließer , 1 = Öffner
      StationsID : DInt;   // Stations ID
      DeviceID : DInt;   // Device ID
   END_VAR
   VAR_OUTPUT
      Error : Bool;   // Fehler
      ErrorState : Byte;   // Fehler Status
      RetVal : DInt;   // Rückgabewert
      "Out-FLTInfo" : "UDTFltFbStructSeqSK";
   END_VAR
   VAR_IN_OUT
      Sensor : "UDT_T_Sensor";   // Datenstruktur vom Sensor
   END_VAR
   VAR
      Save : Bool;
      IEC_Time : TON_TIME;
      IEC_Timer_1 : TON_TIME;
      IEC_Timer_Error : TON_TIME;
   END_VAR
   VAR_TEMP
      TempFrei : Bool;
      Temperror : Bool;
      TempSens : "UDT_T_Sensor";
   END_VAR
   VAR CONSTANT
      cFLT_Busy : DInt := 120;   // Nicht belegt
      cFLT_Free : DInt := 121;   // Nicht frei
      cOK : DInt := 0;
      cFLT_STD_FB_Sensor : DInt := 100000;
   END_VAR
BEGIN

   REGION Read Data

       #TempSens := #Sensor;

   END_REGION
   // Fehlerauswertung Sensor

   #Temperror := #TempSens.Temp_Fehler.Nicht_frei OR #TempSens.Temp_Fehler.Nicht_belegt;
   #IEC_Timer_Error(IN := #Temperror,
             PT := t#5s);

   // fehler Sensor
   #Temperror := (#TempSens.Temp_Fehler.Nicht_frei OR #TempSens.Temp_Fehler.Nicht_belegt)
   AND #IEC_Timer_Error.Q;
   #TempSens.Fehler := #Temperror;
   #Error := #Temperror;

   // Fehlercode Sensor nicht im Sollzustand
   REGION State Sensor
   IF #TempSens.Temp_Fehler.Nicht_frei THEN
       #TempSens.Status := 1;
   ELSIF #TempSens.Temp_Fehler.Nicht_belegt THEN
       #TempSens.Status := 2;
   ELSE
       #TempSens.Status := 0;
   END_IF;
   #ErrorState := #TempSens.Status;


   IF #TempSens.Status <> 0 THEN

       #"Out-FLTInfo".Msg := 1;
       #"Out-FLTInfo".DeviceID := #DeviceID;
       #"Out-FLTInfo".Station := #StationsID;
       IF #TempSens.Status = 1 THEN
           #"Out-FLTInfo".FltID := #cFLT_Free;
       ELSIF #TempSens.Status = 2 THEN
           #"Out-FLTInfo".FltID := #cFLT_Busy;
       END_IF;

   ELSE
       #"Out-FLTInfo".Msg := 0;
       #"Out-FLTInfo".FltID := #cOK;
   END_IF;



   END_REGION

   REGION RetVal Value Output
       IF #TempSens.Status = 0 THEN
           #RetVal := #cOK;
       ELSE
           #RetVal := #cFLT_STD_FB_Sensor;
       END_IF;
   END_REGION

   // Sensor Auswertung

   // Init
   #TempSens.Temp_Fehler.Nicht_frei := False;
   #TempSens.Temp_Fehler.Nicht_belegt := False;
   #TempFrei := #E_Sensor XOR NOT #SensorMode;
   #TempSens.Frei := #TempFrei;
   #TempSens.Belegt := NOT #TempFrei;
   #TempSens.Setup.Typ := #SensorMode;


   IF #TempFrei XOR #Save THEN
       #Save := #TempFrei;
       #IEC_Time(IN := false,
                 PT := t#0ms);
       #IEC_Timer_1(IN:=false,
                    PT:=t#0ms);
       #TempSens.T_Frei := false;
       #TempSens.T_Belegt := False;
       #TempSens.T_Dauer_Belegt := false;


   END_IF;



   IF #TempFrei THEN
       #TempSens.T_Belegt := False;
       #TempSens.T_Dauer_Belegt := false;
       #IEC_Time(IN := #TempFrei,
                 PT := #TempSens.Setup.T_Frei);
       #TempSens.T_Frei := #IEC_Time.Q;
       REGION Reset Timer, wenn Timer nicht neue Zeit hat
           IF #IEC_Time.PT <> #TempSens.Setup.T_Frei THEN
               RESET_TIMER(#IEC_Time);
           END_IF;
       END_REGION
   ELSIF NOT #TempFrei THEN
       #TempSens.T_Frei := False;
       #IEC_Time(IN := NOT #TempFrei,
                 PT := #TempSens.Setup.T_Belegt);
       #IEC_Timer_1(IN := NOT #TempFrei,
                    PT := #TempSens.Setup.T_Dauer);
       #TempSens.T_Belegt := #IEC_Time.Q;
       #TempSens.T_Dauer_Belegt := #IEC_Timer_1.Q;
       REGION Reset Timer, wenn Timer nicht neue Zeit hat
           IF #IEC_Time.PT <> #TempSens.Setup.T_Belegt THEN
               RESET_TIMER(#IEC_Time);
           END_IF;
           IF #IEC_Timer_1.PT <> #TempSens.Setup.T_Dauer THEN
               RESET_TIMER(#IEC_Timer_1);
           END_IF;
       END_REGION
   END_IF;

   REGION Rohsignal
       #TempSens.Rohsignal := #E_Sensor;
   END_REGION

   REGION Write Data

       #Sensor :=#TempSens;

   END_REGION
END_FUNCTION_BLOCK